# EPICS autosave request: iocBoot/gmca_23i_ioc2/dbSave/PIN_St_.req
%
% BURT Request File
%
% $(P)PIN:St: Pin Diode Support
%

file assy.req ASSY=$(P)PIN:St
file mtr1.req MTR1=$(P)PIN:mp
file drv1.req DRV1=$(P)PIN:P

$(P)PIN:P:RqsPosMem1
$(P)PIN:P:RqsPosMem2
